Universal Robots PolyScope program: albin.urp

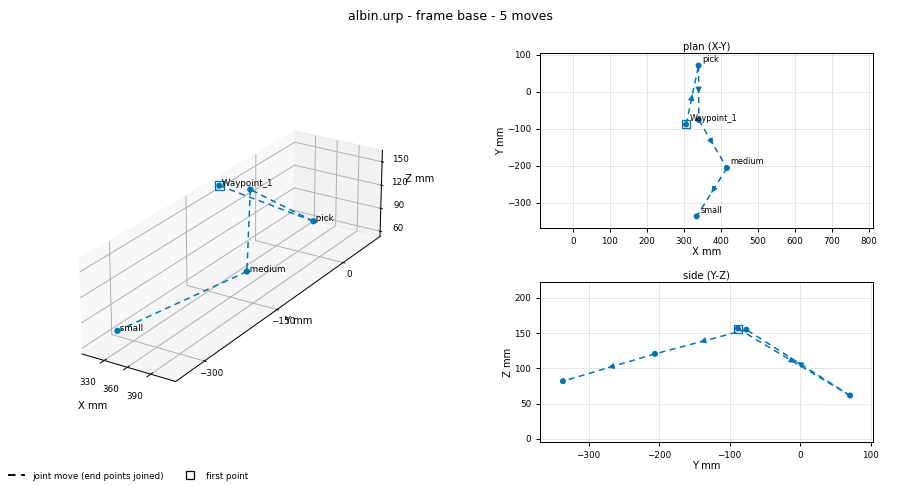
[picture p0: tool path of albin.urp in frame base, 5 of 5 moves have a stored position in this frame; points joined in program order, loops and branches not executed]
Program albin (installation=default directory=/programs/usbdisk createdIn=3.15.7.106331 lastSavedIn=3.15.7.106331 robotSerialNumber=2022330232)
Calibrated DH parameters: a=[-0.000133, -0.226834, -0.203945, 0.000012, -0.000044, 0]; d=[0.151902, -59.477767, 71.768534, -12.178468, 0.085353, 0.082277]; alpha=[1.571593, 0.0015, 0.005101, 1.571815, -1.570835, 0]; deltaTheta=[0.000073, -0.374784, 0.673098, -0.298294, -0.000045, 0.000021]
Robot Program (runOnlyOnce=false)
  MoveJ speed 60 deg/s, acceleration 80 deg/s^2 (useActiveTCP=true)
    Waypoint Waypoint_1: TCP in base x=306.095 y=-88.176 z=156.432 mm, rx=-2.5741 ry=1.7639 rz=0.009 rad; joints [3.954, -91.415, -103.03, -75.065, 91.436, 342.773] deg; flange x=305.345 y=-90.345 z=261.407 mm, rx=-2.5741 ry=1.7639 rz=0.009 rad
  MoveJ speed 60 deg/s, acceleration 80 deg/s^2 (useActiveTCP=true)
    Waypoint pick: TCP in base x=339.846 y=70.89 z=61.456 mm, rx=-2.04 ry=1.8987 rz=0.8293 rad; joints [12.726, -120.055, -100.057, -58.278, 125.095, 366.065] deg; flange x=365.401 y=15.235 z=146.746 mm, rx=-2.04 ry=1.8987 rz=0.8293 rad
  MoveJ speed 60 deg/s, acceleration 80 deg/s^2 (useActiveTCP=true)
    Waypoint Waypoint_3: TCP in base x=340.414 y=-76.134 z=154.956 mm, rx=-2.1805 ry=2.1898 rz=-0.0837 rad; joints [6.63, -96.104, -100.048, -69.669, 89.639, 366.85] deg; flange x=332.677 y=-75.825 z=259.67 mm, rx=-2.1805 ry=2.1898 rz=-0.0837 rad
  MoveJ speed 60 deg/s, acceleration 80 deg/s^2 (useActiveTCP=true)
    Waypoint medium: TCP in base x=416.371 y=-205.929 z=120.574 mm, rx=-1.7512 ry=2.4446 rz=-0.2345 rad; joints [-12.007, -121.894, -77.909, -58.77, 89.633, 366.779] deg; flange x=396.285 y=-200.373 z=223.485 mm, rx=-1.7512 ry=2.4446 rz=-0.2345 rad
  MoveJ speed 60 deg/s, acceleration 80 deg/s^2 (useActiveTCP=true)
    Waypoint small: TCP in base x=334.771 y=-336.499 z=81.831 mm, rx=-1.3025 ry=2.7077 rz=-0.2239 rad; joints [-32.129, -128.401, -77.907, -52.55, 92.009, 366.783] deg; flange x=315.951 y=-328.352 z=184.809 mm, rx=-1.3025 ry=2.7077 rz=-0.2239 rad
